{attribute 'qualified_only' := ''}
{attribute 'strict' := ''}
TYPE cTraySize :
(
	NoSize := 0,
	Small := 1,
	Large := 2
) DINT;
END_TYPE

(* stored: Version 1.1.0.1, ProductVersion 3.1.4024.6
   DUT cTraySize: Id {44e81ab8-c622-4bea-9889-46306b0016ed} *)
